DATA_BLOCK "Keep_DB"
{ S7_Optimized_Access := 'FALSE' }
VERSION : 0.1
VAR RETAIN
      Ana_Keep : Array[1..40] of "UDT_Ana_Keep";   // 模拟量保持数据数组[1..40]

      Device_Keep : Array[1..10] of "UDT_Device_Keep";   // 设备控制保持数据数组[1..10]

      Valve_Keep : Array[1..15] of "UDT_Valve_Keep";   // 阀门控制保持数据数组[1..15]
   END_VAR


BEGIN
END_DATA_BLOCK